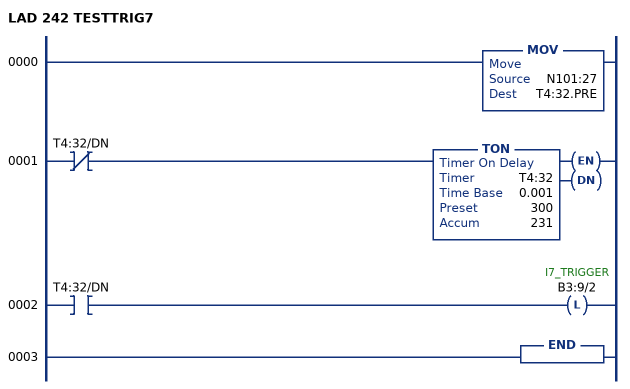
% Rung: 0 %
SOR MOV N101:27 T4:32.PRE EOR
%   N101:27  I7_TRIGTIME %
% Rung: 1 %
SOR XIO T4:32/DN TON T4:32 0.001 300 231 EOR
% Rung: 2 %
SOR XIC T4:32/DN OTL B3:9/2 EOR
%   B3:9/2  I7_TRIGGER %
% Rung: 3 %
SOR END EOR

LADDER 243 "TESTTRIG8"
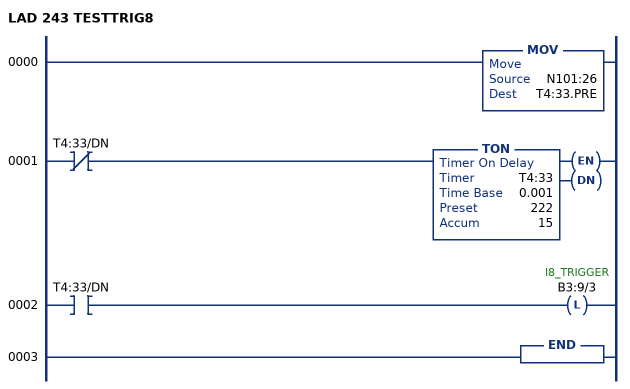
% Rung: 0 %
SOR MOV N101:26 T4:33.PRE EOR
%   N101:26  I8_TRIGTIME %
% Rung: 1 %
SOR XIO T4:33/DN TON T4:33 0.001 222 15 EOR
% Rung: 2 %
SOR XIC T4:33/DN OTL B3:9/3 EOR
%   B3:9/3  I8_TRIGGER %
% Rung: 3 %
SOR END EOR

LADDER 244 "PACKAGER"    % normal %
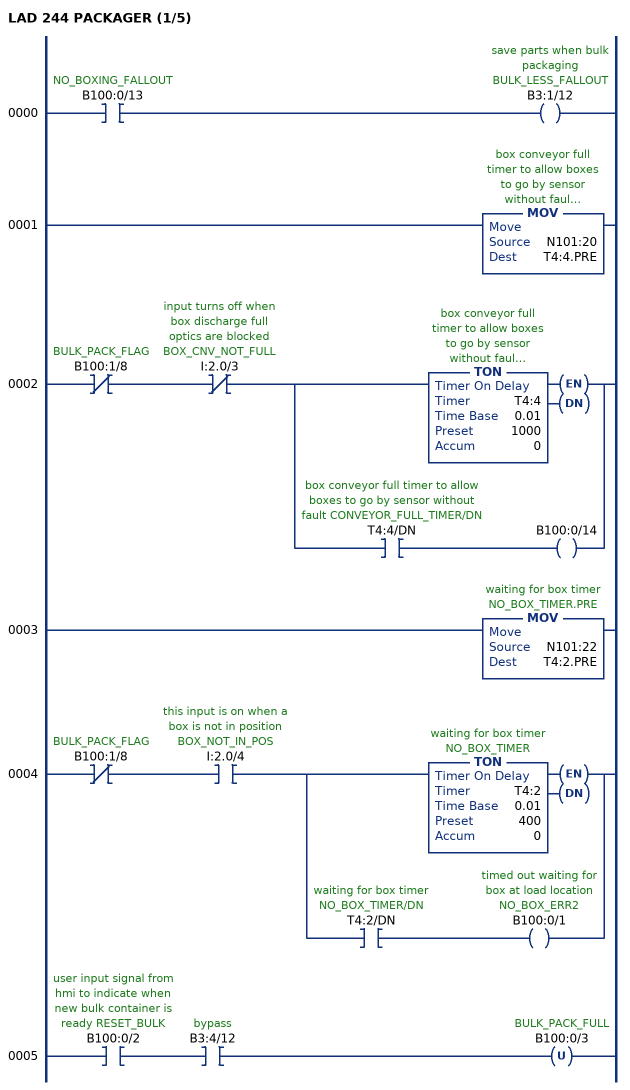
% Rung: 0 %
SOR XIC B100:0/13 OTE B3:1/12 EOR
%   B100:0/13  NO_BOXING_FALLOUT %
%   B3:1/12  BULK_LESS_FALLOUT  "save parts when bulk packaging" %
% Rung: 1 %
SOR MOV N101:20 T4:4.PRE EOR
%   N101:20  CONV_FULL_TIME_LIMIT  "time to allow box to pass box conveyor full sensor without fault" %
%   T4:4  CONVEYOR_FULL_TIMER  "box conveyor full timer to allow boxes to go by sensor without fault" %
% Rung: 2 %
SOR XIO B100:1/8 XIO I:2.0/3 BST TON T4:4 0.01 1000 0 NXB XIC T4:4/DN OTE B100:0/14 BND EOR
%   B100:1/8  BULK_PACK_FLAG %
%   I:2.0/3  BOX_CNV_NOT_FULL  "input turns off when box discharge full optics are blocked" %
%   T4:4  CONVEYOR_FULL_TIMER  "box conveyor full timer to allow boxes to go by sensor without fault" %
% Rung: 3 %
SOR MOV N101:22 T4:2.PRE EOR
%   N101:22  BOX_WAIT_TIME_LIMIT  "the time until waiting for box message in hmi (fault)" %
%   T4:2  NO_BOX_TIMER  "waiting for box timer" %
% Rung: 4 %
SOR XIO B100:1/8 XIC I:2.0/4 BST TON T4:2 0.01 400 0 NXB XIC T4:2/DN OTE B100:0/1 BND EOR
%   B100:1/8  BULK_PACK_FLAG %
%   I:2.0/4  BOX_NOT_IN_POS  "this input is on when a box is not in position" %
%   T4:2  NO_BOX_TIMER  "waiting for box timer" %
%   B100:0/1  NO_BOX_ERR2  "timed out waiting for box at load location" %
% Rung: 5 %
SOR XIC B100:0/2 XIC B3:4/12 OTU B100:0/3 EOR
%   B100:0/2  RESET_BULK  "user input signal from hmi to indicate when new bulk container is ready" %
%   B3:4/12  "bypass" %
%   B100:0/3  BULK_PACK_FULL %

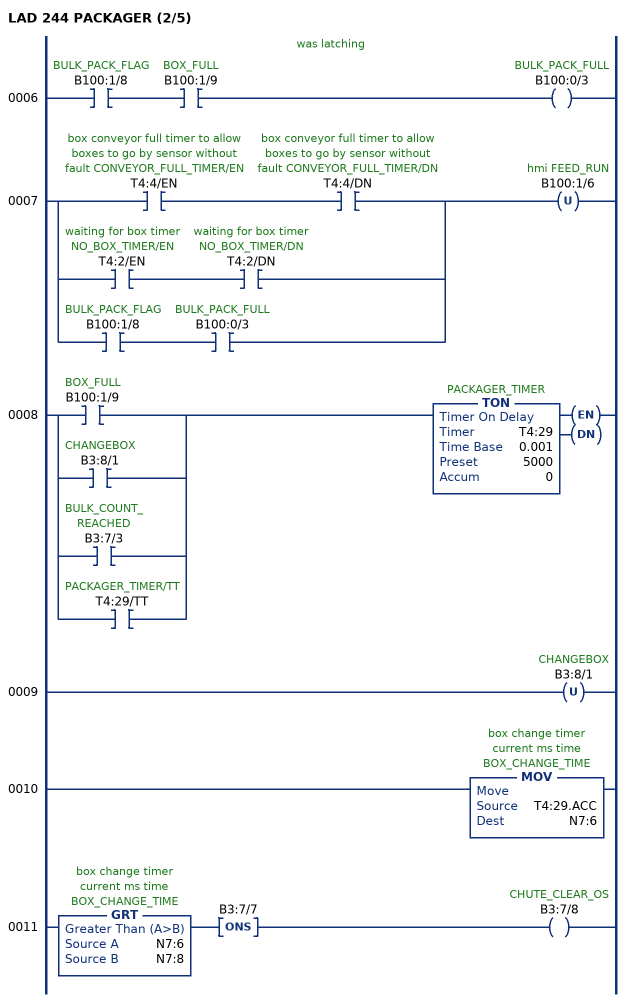
% Rung: 6 %
% was latching %
SOR XIC B100:1/8 XIC B100:1/9 OTE B100:0/3 EOR
%   B100:1/8  BULK_PACK_FLAG %
%   B100:1/9  BOX_FULL %
%   B100:0/3  BULK_PACK_FULL %
% Rung: 7 %
SOR BST XIC T4:4/EN XIC T4:4/DN NXB XIC T4:2/EN XIC T4:2/DN NXB XIC B100:1/8 XIC B100:0/3 BND OTU B100:1/6 EOR
%   T4:4  CONVEYOR_FULL_TIMER  "box conveyor full timer to allow boxes to go by sensor without fault" %
%   T4:2  NO_BOX_TIMER  "waiting for box timer" %
%   B100:1/8  BULK_PACK_FLAG %
%   B100:0/3  BULK_PACK_FULL %
%   B100:1/6  FEED_RUN  "hmi" %
% Rung: 8 %
SOR BST XIC B100:1/9 NXB XIC B3:8/1 NXB XIC B3:7/3 NXB XIC T4:29/TT BND TON T4:29 0.001 5000 0 EOR
%   B100:1/9  BOX_FULL %
%   B3:8/1  CHANGEBOX %
%   B3:7/3  BULK_COUNT_REACHED %
%   T4:29  PACKAGER_TIMER %
% Rung: 9 %
SOR OTU B3:8/1 EOR
%   B3:8/1  CHANGEBOX %
% Rung: 10 %
SOR MOV T4:29.ACC N7:6 EOR
%   T4:29  PACKAGER_TIMER %
%   N7:6  BOX_CHANGE_TIME  "box change timer current ms time" %
% Rung: 11 %
SOR GRT N7:6 N7:8 ONS B3:7/7 OTE B3:7/8 EOR
%   N7:6  BOX_CHANGE_TIME  "box change timer current ms time" %
%   N7:8  CHUTE_CLEAR_TIME %
%   B3:7/8  CHUTE_CLEAR_OS %

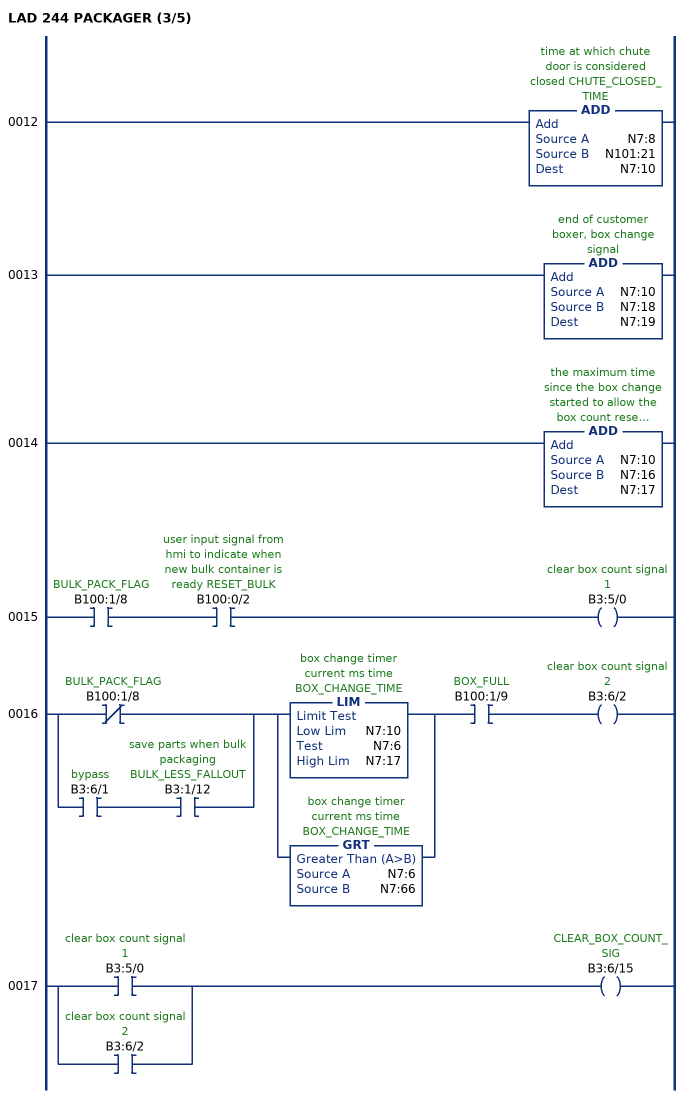
% Rung: 12 %
SOR ADD N7:8 N101:21 N7:10 EOR
%   N7:8  CHUTE_CLEAR_TIME %
%   N101:21  CHUTE_CLOSE_TIME  "ms time required to close chute" %
%   N7:10  CHUTE_CLOSED_TIME  "time at which chute door is considered closed" %
% Rung: 13 %
SOR ADD N7:10 N7:18 N7:19 EOR
%   N7:10  CHUTE_CLOSED_TIME  "time at which chute door is considered closed" %
%   N7:18  CHANGE_BOX_SIG_TIME  "customer boxer change box signal time" %
%   N7:19  "end of customer boxer, box change signal" %
% Rung: 14 %
SOR ADD N7:10 N7:16 N7:17 EOR
%   N7:10  CHUTE_CLOSED_TIME  "time at which chute door is considered closed" %
%   N7:16  RESET_COUNT_SIG_TIME  "maximum length of time to hold box count reset signal on" %
%   N7:17  "the maximum time since the box change started to allow the box count reset signal" %
% Rung: 15 %
SOR XIC B100:1/8 XIC B100:0/2 OTE B3:5/0 EOR
%   B100:1/8  BULK_PACK_FLAG %
%   B100:0/2  RESET_BULK  "user input signal from hmi to indicate when new bulk container is ready" %
%   B3:5/0  "clear box count signal 1" %
% Rung: 16 %
SOR BST XIO B100:1/8 NXB XIC B3:6/1 XIC B3:1/12 BND BST LIM N7:10 N7:6 N7:17 NXB GRT N7:6 N7:66 BND XIC B100:1/9 OTE B3:6/2 EOR
%   B100:1/8  BULK_PACK_FLAG %
%   B3:6/1  "bypass" %
%   B3:1/12  BULK_LESS_FALLOUT  "save parts when bulk packaging" %
%   N7:10  CHUTE_CLOSED_TIME  "time at which chute door is considered closed" %
%   N7:6  BOX_CHANGE_TIME  "box change timer current ms time" %
%   N7:17  "the maximum time since the box change started to allow the box count reset signal" %
%   B100:1/9  BOX_FULL %
%   B3:6/2  "clear box count signal 2" %
% Rung: 17 %
SOR BST XIC B3:5/0 NXB XIC B3:6/2 BND OTE B3:6/15 EOR
%   B3:5/0  "clear box count signal 1" %
%   B3:6/2  "clear box count signal 2" %
%   B3:6/15  CLEAR_BOX_COUNT_SIG %

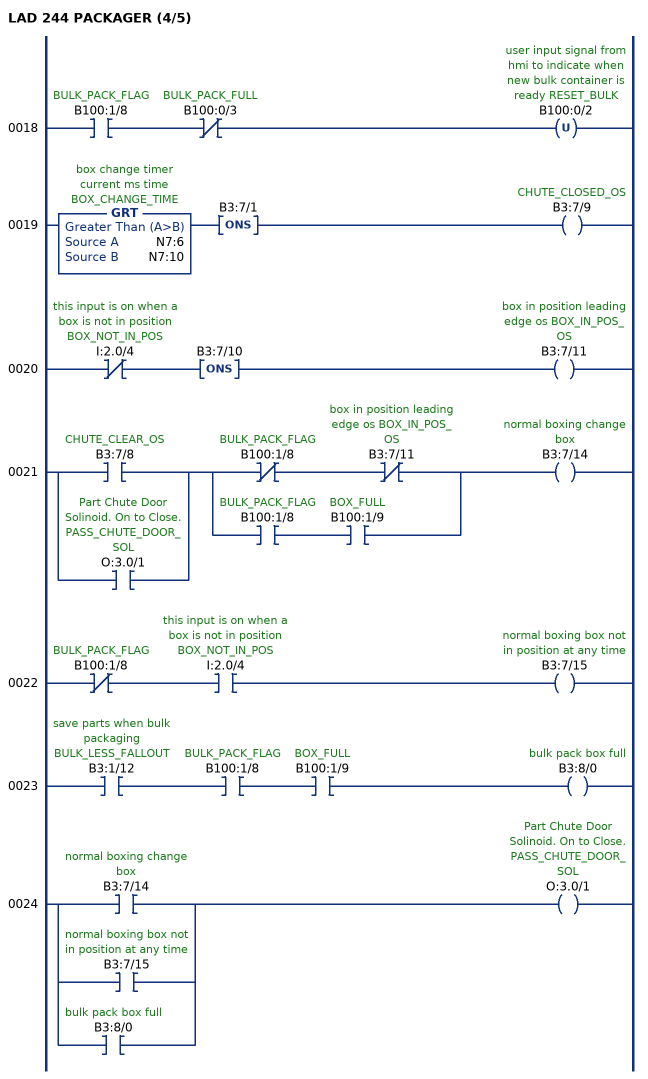
% Rung: 18 %
SOR XIC B100:1/8 XIO B100:0/3 OTU B100:0/2 EOR
%   B100:1/8  BULK_PACK_FLAG %
%   B100:0/3  BULK_PACK_FULL %
%   B100:0/2  RESET_BULK  "user input signal from hmi to indicate when new bulk container is ready" %
% Rung: 19 %
SOR GRT N7:6 N7:10 ONS B3:7/1 OTE B3:7/9 EOR
%   N7:6  BOX_CHANGE_TIME  "box change timer current ms time" %
%   N7:10  CHUTE_CLOSED_TIME  "time at which chute door is considered closed" %
%   B3:7/9  CHUTE_CLOSED_OS %
% Rung: 20 %
SOR XIO I:2.0/4 ONS B3:7/10 OTE B3:7/11 EOR
%   I:2.0/4  BOX_NOT_IN_POS  "this input is on when a box is not in position" %
%   B3:7/11  BOX_IN_POS_OS  "box in position leading edge os" %
% Rung: 21 %
SOR BST XIC B3:7/8 NXB XIC O:3.0/1 BND BST XIO B100:1/8 XIO B3:7/11 NXB XIC B100:1/8 XIC B100:1/9 BND OTE B3:7/14 EOR
%   B3:7/8  CHUTE_CLEAR_OS %
%   O:3.0/1  PASS_CHUTE_DOOR_SOL  "Part Chute Door Solinoid. On to Close." %
%   B100:1/8  BULK_PACK_FLAG %
%   B3:7/11  BOX_IN_POS_OS  "box in position leading edge os" %
%   B100:1/9  BOX_FULL %
%   B3:7/14  "normal boxing change box" %
% Rung: 22 %
SOR XIO B100:1/8 XIC I:2.0/4 OTE B3:7/15 EOR
%   B100:1/8  BULK_PACK_FLAG %
%   I:2.0/4  BOX_NOT_IN_POS  "this input is on when a box is not in position" %
%   B3:7/15  "normal boxing box not in position at any time" %
% Rung: 23 %
SOR XIC B3:1/12 XIC B100:1/8 XIC B100:1/9 OTE B3:8/0 EOR
%   B3:1/12  BULK_LESS_FALLOUT  "save parts when bulk packaging" %
%   B100:1/8  BULK_PACK_FLAG %
%   B100:1/9  BOX_FULL %
%   B3:8/0  "bulk pack box full" %
% Rung: 24 %
SOR BST XIC B3:7/14 NXB XIC B3:7/15 NXB XIC B3:8/0 BND OTE O:3.0/1 EOR
%   B3:7/14  "normal boxing change box" %
%   B3:7/15  "normal boxing box not in position at any time" %
%   B3:8/0  "bulk pack box full" %
%   O:3.0/1  PASS_CHUTE_DOOR_SOL  "Part Chute Door Solinoid. On to Close." %

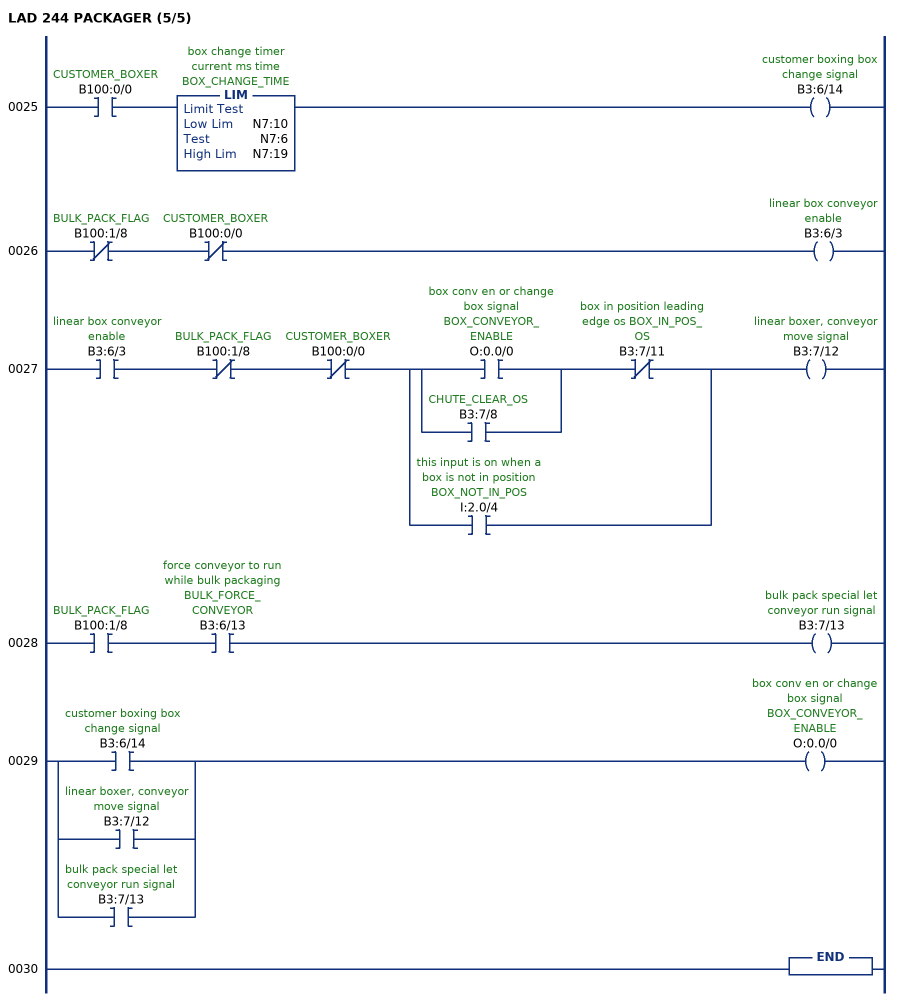
% Rung: 25 %
SOR XIC B100:0/0 LIM N7:10 N7:6 N7:19 OTE B3:6/14 EOR
%   B100:0/0  CUSTOMER_BOXER %
%   N7:10  CHUTE_CLOSED_TIME  "time at which chute door is considered closed" %
%   N7:6  BOX_CHANGE_TIME  "box change timer current ms time" %
%   N7:19  "end of customer boxer, box change signal" %
%   B3:6/14  "customer boxing box change signal" %
% Rung: 26 %
SOR XIO B100:1/8 XIO B100:0/0 OTE B3:6/3 EOR
%   B100:1/8  BULK_PACK_FLAG %
%   B100:0/0  CUSTOMER_BOXER %
%   B3:6/3  "linear box conveyor enable" %
% Rung: 27 %
SOR XIC B3:6/3 XIO B100:1/8 XIO B100:0/0 BST BST XIC O:0.0/0 NXB XIC B3:7/8 BND XIO B3:7/11 NXB XIC I:2.0/4 BND OTE B3:7/12 EOR
%   B3:6/3  "linear box conveyor enable" %
%   B100:1/8  BULK_PACK_FLAG %
%   B100:0/0  CUSTOMER_BOXER %
%   O:0.0/0  BOX_CONVEYOR_ENABLE  "box conv en or change box signal" %
%   B3:7/8  CHUTE_CLEAR_OS %
%   B3:7/11  BOX_IN_POS_OS  "box in position leading edge os" %
%   I:2.0/4  BOX_NOT_IN_POS  "this input is on when a box is not in position" %
%   B3:7/12  "linear boxer, conveyor move signal" %
% Rung: 28 %
SOR XIC B100:1/8 XIC B3:6/13 OTE B3:7/13 EOR
%   B100:1/8  BULK_PACK_FLAG %
%   B3:6/13  BULK_FORCE_CONVEYOR  "force conveyor to run while bulk packaging" %
%   B3:7/13  "bulk pack special let conveyor run signal" %
% Rung: 29 %
SOR BST XIC B3:6/14 NXB XIC B3:7/12 NXB XIC B3:7/13 BND OTE O:0.0/0 EOR
%   B3:6/14  "customer boxing box change signal" %
%   B3:7/12  "linear boxer, conveyor move signal" %
%   B3:7/13  "bulk pack special let conveyor run signal" %
%   O:0.0/0  BOX_CONVEYOR_ENABLE  "box conv en or change box signal" %
% Rung: 30 %
SOR END EOR

LADDER 245 "NO PACKAGE"
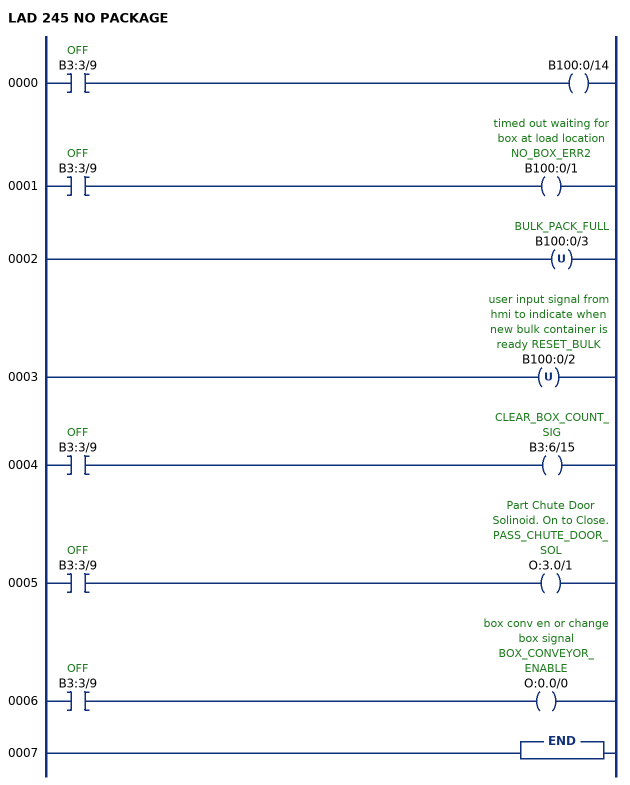
% Rung: 0 %
SOR XIC B3:3/9 OTE B100:0/14 EOR
%   B3:3/9  OFF %
% Rung: 1 %
SOR XIC B3:3/9 OTE B100:0/1 EOR
%   B3:3/9  OFF %
%   B100:0/1  NO_BOX_ERR2  "timed out waiting for box at load location" %
% Rung: 2 %
SOR OTU B100:0/3 EOR
%   B100:0/3  BULK_PACK_FULL %
% Rung: 3 %
SOR OTU B100:0/2 EOR
%   B100:0/2  RESET_BULK  "user input signal from hmi to indicate when new bulk container is ready" %
% Rung: 4 %
SOR XIC B3:3/9 OTE B3:6/15 EOR
%   B3:3/9  OFF %
%   B3:6/15  CLEAR_BOX_COUNT_SIG %
% Rung: 5 %
SOR XIC B3:3/9 OTE O:3.0/1 EOR
%   B3:3/9  OFF %
%   O:3.0/1  PASS_CHUTE_DOOR_SOL  "Part Chute Door Solinoid. On to Close." %
% Rung: 6 %
SOR XIC B3:3/9 OTE O:0.0/0 EOR
%   B3:3/9  OFF %
%   O:0.0/0  BOX_CONVEYOR_ENABLE  "box conv en or change box signal" %
% Rung: 7 %
SOR END EOR

LADDER 246 "RATE1"
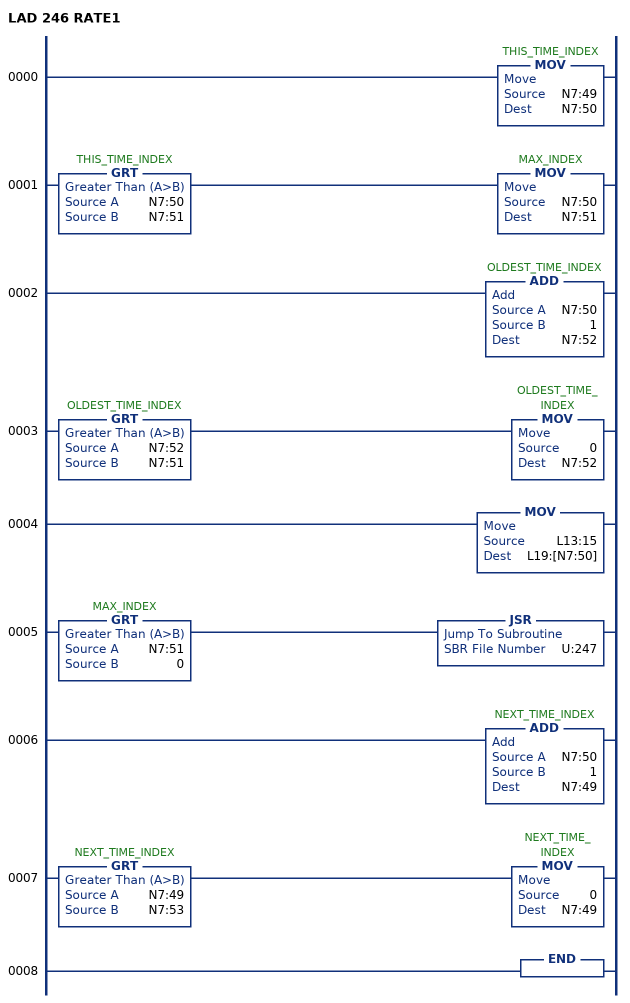
% Rung: 0 %
SOR MOV N7:49 N7:50 EOR
%   N7:49  NEXT_TIME_INDEX %
%   N7:50  THIS_TIME_INDEX %
% Rung: 1 %
SOR GRT N7:50 N7:51 MOV N7:50 N7:51 EOR
%   N7:50  THIS_TIME_INDEX %
%   N7:51  MAX_INDEX %
% Rung: 2 %
SOR ADD N7:50 1 N7:52 EOR
%   N7:50  THIS_TIME_INDEX %
%   N7:52  OLDEST_TIME_INDEX %
% Rung: 3 %
SOR GRT N7:52 N7:51 MOV 0 N7:52 EOR
%   N7:52  OLDEST_TIME_INDEX %
%   N7:51  MAX_INDEX %
% Rung: 4 %
SOR MOV L13:15 L19:[N7:50] EOR
%   L13:15  THE_TIME %
%   N7:50  THIS_TIME_INDEX %
% Rung: 5 %
SOR GRT N7:51 0 JSR U:247 EOR
%   N7:51  MAX_INDEX %
% Rung: 6 %
SOR ADD N7:50 1 N7:49 EOR
%   N7:50  THIS_TIME_INDEX %
%   N7:49  NEXT_TIME_INDEX %
% Rung: 7 %
SOR GRT N7:49 N7:53 MOV 0 N7:49 EOR
%   N7:49  NEXT_TIME_INDEX %
%   N7:53  UPPER_INDEX_LIMIT %
% Rung: 8 %
SOR END EOR

LADDER 247 "RATE2"
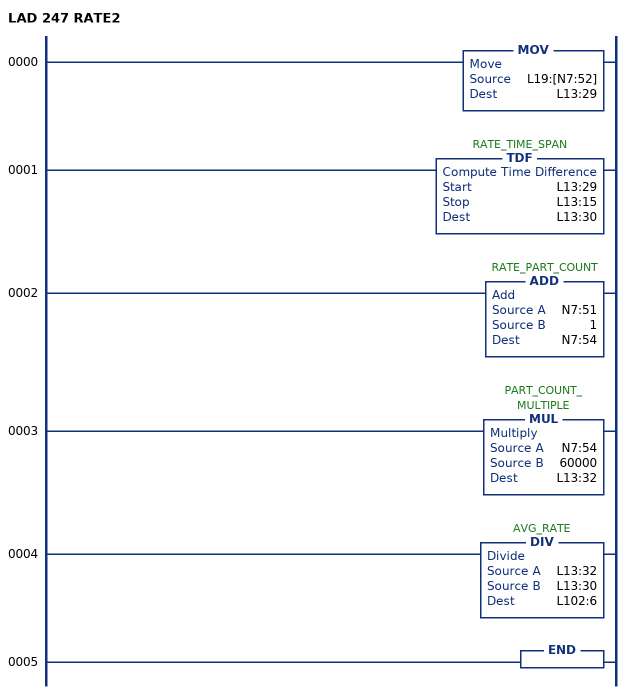
% Rung: 0 %
SOR MOV L19:[N7:52] L13:29 EOR
%   N7:52  OLDEST_TIME_INDEX %
% Rung: 1 %
SOR TDF L13:29 L13:15 L13:30 EOR
%   L13:15  THE_TIME %
%   L13:30  RATE_TIME_SPAN %
% Rung: 2 %
SOR ADD N7:51 1 N7:54 EOR
%   N7:51  MAX_INDEX %
%   N7:54  RATE_PART_COUNT %
% Rung: 3 %
SOR MUL N7:54 60000 L13:32 EOR
%   N7:54  RATE_PART_COUNT %
%   L13:32  PART_COUNT_MULTIPLE %
% Rung: 4 %
SOR DIV L13:32 L13:30 L102:6 EOR
%   L13:32  PART_COUNT_MULTIPLE %
%   L13:30  RATE_TIME_SPAN %
%   L102:6  AVG_RATE %
% Rung: 5 %
SOR END EOR

LADDER 248 "RESET RATE"
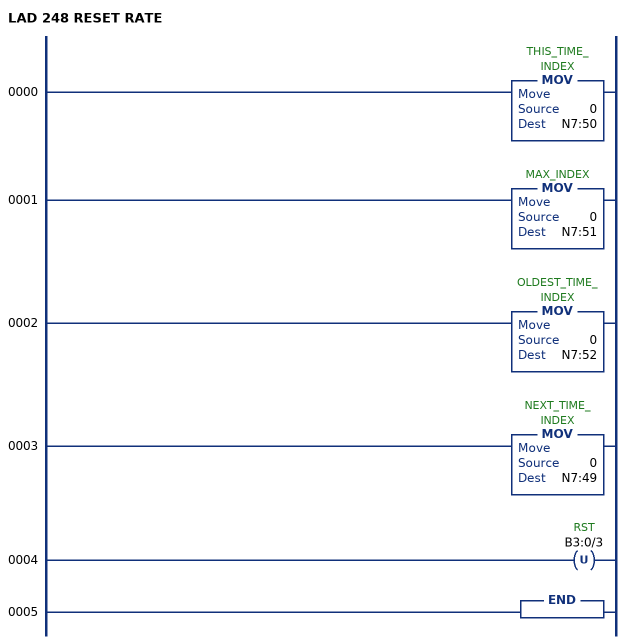
% Rung: 0 %
SOR MOV 0 N7:50 EOR
%   N7:50  THIS_TIME_INDEX %
% Rung: 1 %
SOR MOV 0 N7:51 EOR
%   N7:51  MAX_INDEX %
% Rung: 2 %
SOR MOV 0 N7:52 EOR
%   N7:52  OLDEST_TIME_INDEX %
% Rung: 3 %
SOR MOV 0 N7:49 EOR
%   N7:49  NEXT_TIME_INDEX %
% Rung: 4 %
SOR OTU B3:0/3 EOR
%   B3:0/3  RST %
% Rung: 5 %
SOR END EOR

LADDER 249 "NP STOP"    % stop on no good %
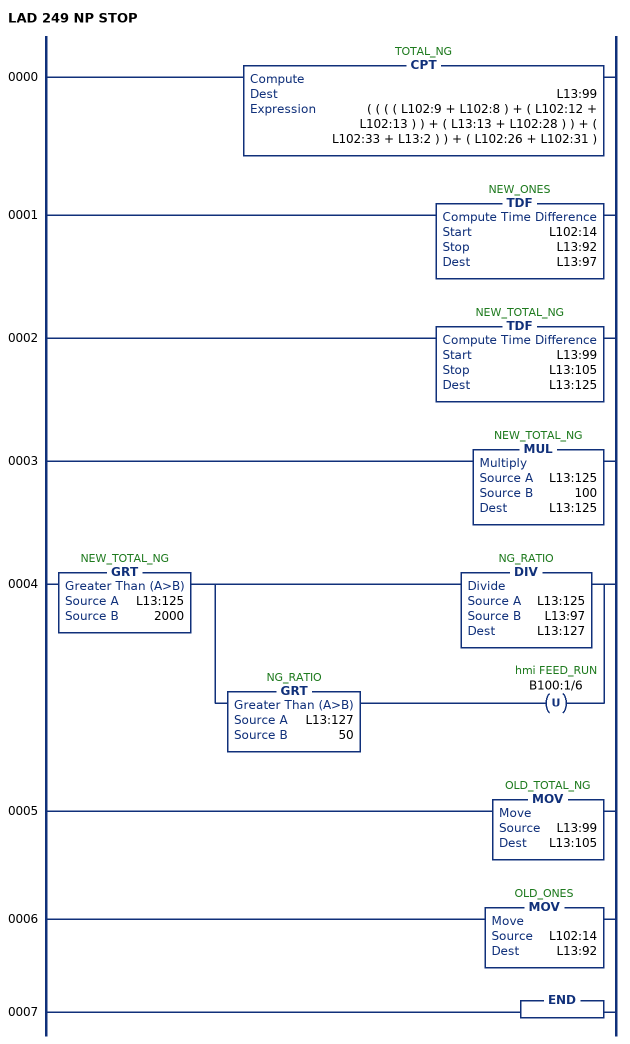
% Rung: 0 %
SOR CPT L13:99 " ( ( ( ( L102:9 + L102:8 ) + ( L102:12 + L102:13 ) ) + ( L13:13 + L102:28 ) ) + ( L102:33 + L13:2 ) ) + ( L102:26 + L102:31 ) " EOR
%   L13:99  TOTAL_NG %
%   L102:9  "too wide bottom" %
%   L102:8  "too close bottom" %
%   L102:12  "too close top count" %
%   L102:13  "too wide top count" %
%   L102:28  I1_I5_SKIPPEDCOUNT %
%   L102:33  I2_I6_SKIPPEDCOUNT %
%   L102:26  I1_I5_FAIL_COUNT %
%   L102:31  I2_I6_FAIL_COUNT %
% Rung: 1 %
SOR TDF L102:14 L13:92 L13:97 EOR
%   L102:14  ONES %
%   L13:92  OLD_ONES %
%   L13:97  NEW_ONES %
% Rung: 2 %
SOR TDF L13:99 L13:105 L13:125 EOR
%   L13:99  TOTAL_NG %
%   L13:105  OLD_TOTAL_NG %
%   L13:125  NEW_TOTAL_NG %
% Rung: 3 %
SOR MUL L13:125 100 L13:125 EOR
%   L13:125  NEW_TOTAL_NG %
% Rung: 4 %
SOR GRT L13:125 2000 BST DIV L13:125 L13:97 L13:127 NXB GRT L13:127 50 OTU B100:1/6 BND EOR
%   L13:125  NEW_TOTAL_NG %
%   L13:97  NEW_ONES %
%   L13:127  NG_RATIO %
%   B100:1/6  FEED_RUN  "hmi" %
% Rung: 5 %
SOR MOV L13:99 L13:105 EOR
%   L13:99  TOTAL_NG %
%   L13:105  OLD_TOTAL_NG %
% Rung: 6 %
SOR MOV L102:14 L13:92 EOR
%   L102:14  ONES %
%   L13:92  OLD_ONES %
% Rung: 7 %
SOR END EOR

LADDER 250 "SPEED BOT"    % high speed %
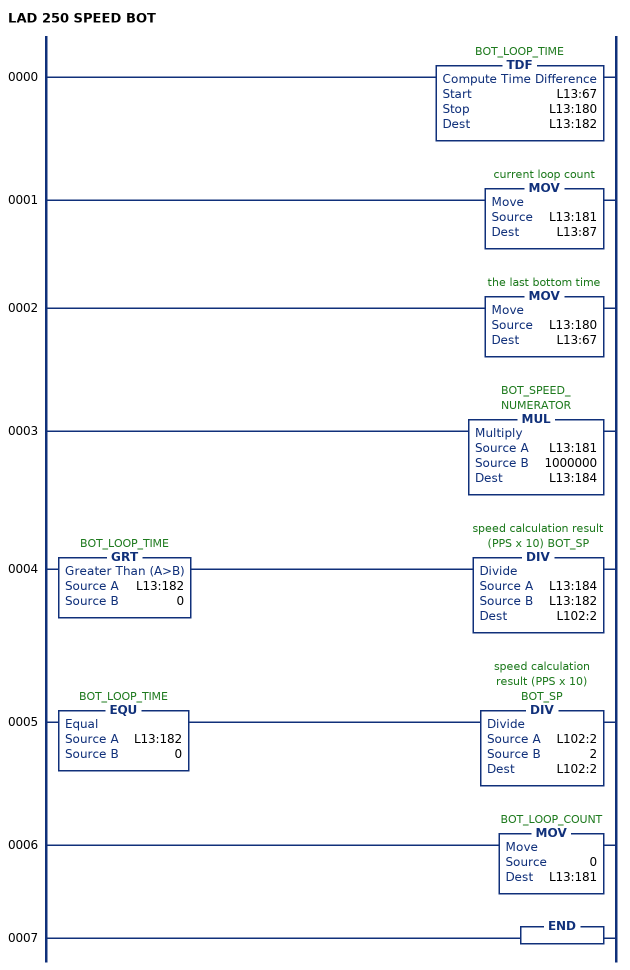
% Rung: 0 %
SOR TDF L13:67 L13:180 L13:182 EOR
%   L13:67  "the last bottom time" %
%   L13:180  BOT_THIS_TIME  "rtc bot belt movement event time" %
%   L13:182  BOT_LOOP_TIME %
% Rung: 1 %
SOR MOV L13:181 L13:87 EOR
%   L13:181  BOT_LOOP_COUNT %
%   L13:87  "current loop count" %
% Rung: 2 %
SOR MOV L13:180 L13:67 EOR
%   L13:180  BOT_THIS_TIME  "rtc bot belt movement event time" %
%   L13:67  "the last bottom time" %
% Rung: 3 %
SOR MUL L13:181 1000000 L13:184 EOR
%   L13:181  BOT_LOOP_COUNT %
%   L13:184  BOT_SPEED_NUMERATOR %
% Rung: 4 %
SOR GRT L13:182 0 DIV L13:184 L13:182 L102:2 EOR
%   L13:182  BOT_LOOP_TIME %
%   L13:184  BOT_SPEED_NUMERATOR %
%   L102:2  BOT_SP  "speed calculation result (PPS x 10)" %
% Rung: 5 %
SOR EQU L13:182 0 DIV L102:2 2 L102:2 EOR
%   L13:182  BOT_LOOP_TIME %
%   L102:2  BOT_SP  "speed calculation result (PPS x 10)" %
% Rung: 6 %
SOR MOV 0 L13:181 EOR
%   L13:181  BOT_LOOP_COUNT %
% Rung: 7 %
SOR END EOR

LADDER 251 "SPEED TOP"    % high speed %
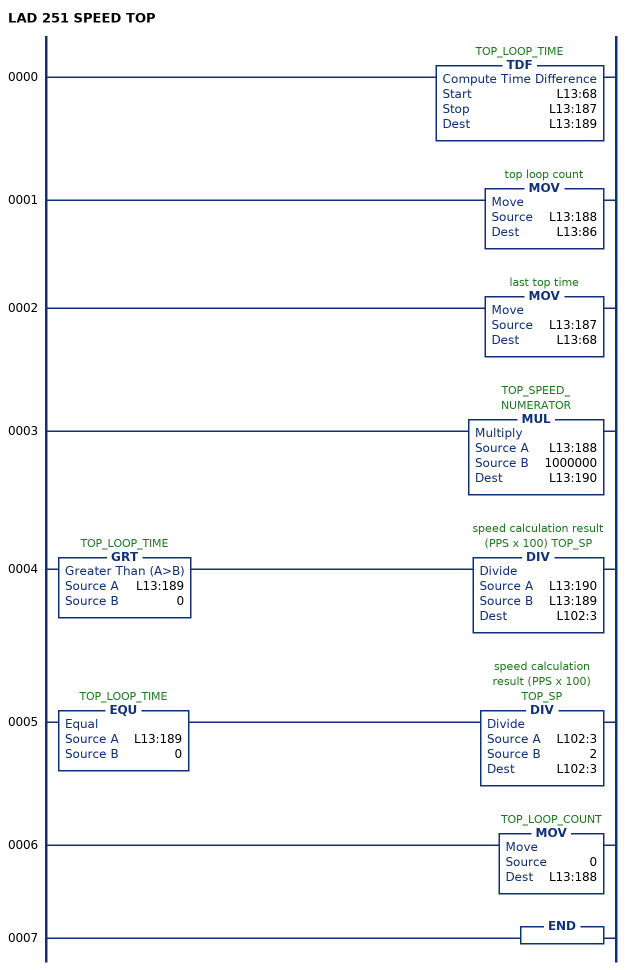
% Rung: 0 %
SOR TDF L13:68 L13:187 L13:189 EOR
%   L13:68  "last top time" %
%   L13:187  TOP_THIS_TIME  "rtc top belt movement event time" %
%   L13:189  TOP_LOOP_TIME %
% Rung: 1 %
SOR MOV L13:188 L13:86 EOR
%   L13:188  TOP_LOOP_COUNT %
%   L13:86  "top loop count" %
% Rung: 2 %
SOR MOV L13:187 L13:68 EOR
%   L13:187  TOP_THIS_TIME  "rtc top belt movement event time" %
%   L13:68  "last top time" %
% Rung: 3 %
SOR MUL L13:188 1000000 L13:190 EOR
%   L13:188  TOP_LOOP_COUNT %
%   L13:190  TOP_SPEED_NUMERATOR %
% Rung: 4 %
SOR GRT L13:189 0 DIV L13:190 L13:189 L102:3 EOR
%   L13:189  TOP_LOOP_TIME %
%   L13:190  TOP_SPEED_NUMERATOR %
%   L102:3  TOP_SP  "speed calculation result (PPS x 100)" %
% Rung: 5 %
SOR EQU L13:189 0 DIV L102:3 2 L102:3 EOR
%   L13:189  TOP_LOOP_TIME %
%   L102:3  TOP_SP  "speed calculation result (PPS x 100)" %
% Rung: 6 %
SOR MOV 0 L13:188 EOR
%   L13:188  TOP_LOOP_COUNT %
% Rung: 7 %
SOR END EOR

LADDER 252 "P BOT"    % high speed %
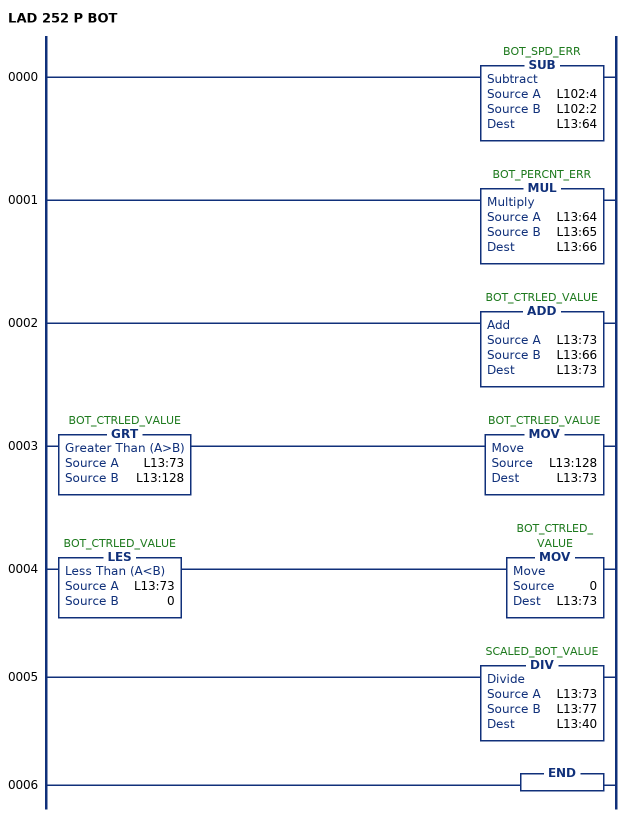
% Rung: 0 %
SOR SUB L102:4 L102:2 L13:64 EOR
%   L102:4  BOT_SPD_SETPOINT %
%   L102:2  BOT_SP  "speed calculation result (PPS x 10)" %
%   L13:64  BOT_SPD_ERR %
% Rung: 1 %
SOR MUL L13:64 L13:65 L13:66 EOR
%   L13:64  BOT_SPD_ERR %
%   L13:65  POS5SHIFT %
%   L13:66  BOT_PERCNT_ERR %
% Rung: 2 %
SOR ADD L13:73 L13:66 L13:73 EOR
%   L13:73  BOT_CTRLED_VALUE %
%   L13:66  BOT_PERCNT_ERR %
% Rung: 3 %
SOR GRT L13:73 L13:128 MOV L13:128 L13:73 EOR
%   L13:73  BOT_CTRLED_VALUE %
%   L13:128  "how much top has shifted since measurment" %
% Rung: 4 %
SOR LES L13:73 0 MOV 0 L13:73 EOR
%   L13:73  BOT_CTRLED_VALUE %
% Rung: 5 %
SOR DIV L13:73 L13:77 L13:40 EOR
%   L13:73  BOT_CTRLED_VALUE %
%   L13:40  SCALED_BOT_VALUE %
% Rung: 6 %
SOR END EOR

LADDER 253 "P TOP"    % high speed %
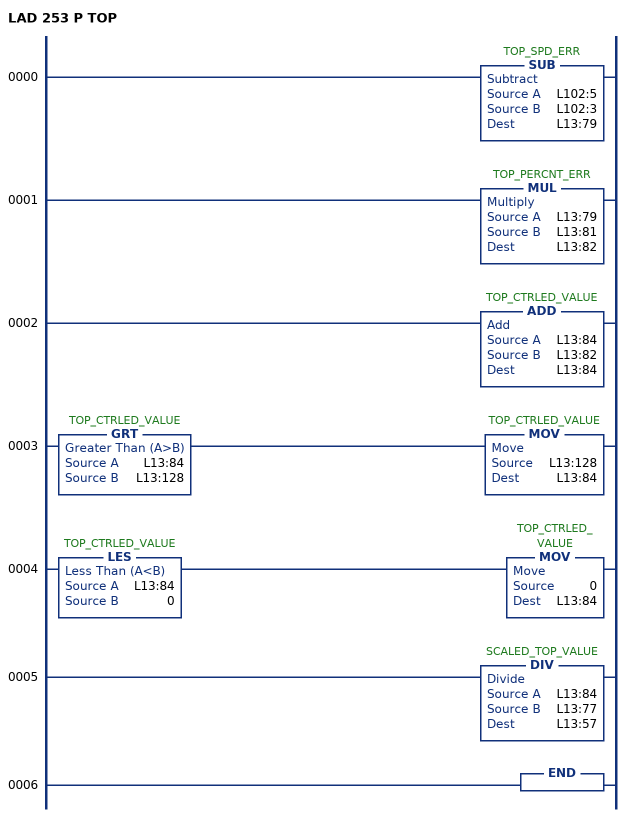
% Rung: 0 %
SOR SUB L102:5 L102:3 L13:79 EOR
%   L102:5  TOP_SPD_SETPOINT %
%   L102:3  TOP_SP  "speed calculation result (PPS x 100)" %
%   L13:79  TOP_SPD_ERR %
% Rung: 1 %
SOR MUL L13:79 L13:81 L13:82 EOR
%   L13:79  TOP_SPD_ERR %
%   L13:81  TOP_FDBK_RATIO %
%   L13:82  TOP_PERCNT_ERR %
% Rung: 2 %
SOR ADD L13:84 L13:82 L13:84 EOR
%   L13:84  TOP_CTRLED_VALUE %
%   L13:82  TOP_PERCNT_ERR %
% Rung: 3 %
SOR GRT L13:84 L13:128 MOV L13:128 L13:84 EOR
%   L13:84  TOP_CTRLED_VALUE %
%   L13:128  "how much top has shifted since measurment" %
% Rung: 4 %
SOR LES L13:84 0 MOV 0 L13:84 EOR
%   L13:84  TOP_CTRLED_VALUE %
% Rung: 5 %
SOR DIV L13:84 L13:77 L13:57 EOR
%   L13:84  TOP_CTRLED_VALUE %
%   L13:57  SCALED_TOP_VALUE %
% Rung: 6 %
SOR END EOR

LADDER 254 "TOTALCOUNT"
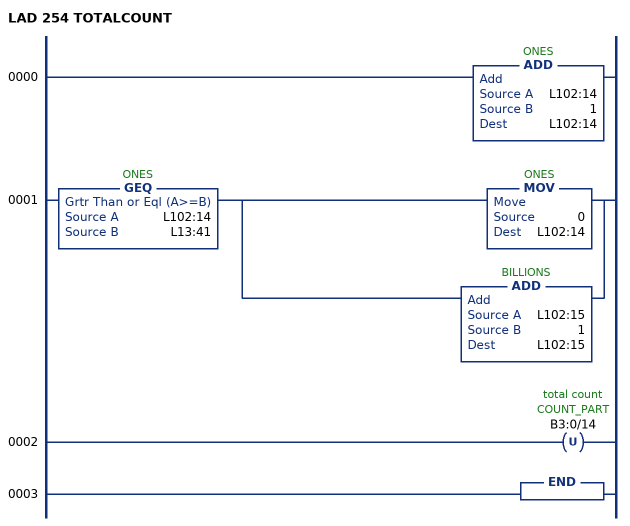
% Rung: 0 %
SOR ADD L102:14 1 L102:14 EOR
%   L102:14  ONES %
% Rung: 1 %
SOR GEQ L102:14 L13:41 BST MOV 0 L102:14 NXB ADD L102:15 1 L102:15 BND EOR
%   L102:14  ONES %
%   L13:41  "skipped count change in the last 3 seconds" %
%   L102:15  BILLIONS %
% Rung: 2 %
SOR OTU B3:0/14 EOR
%   B3:0/14  COUNT_PART  "total count" %
% Rung: 3 %
SOR END EOR

LADDER 255 "SAVED"
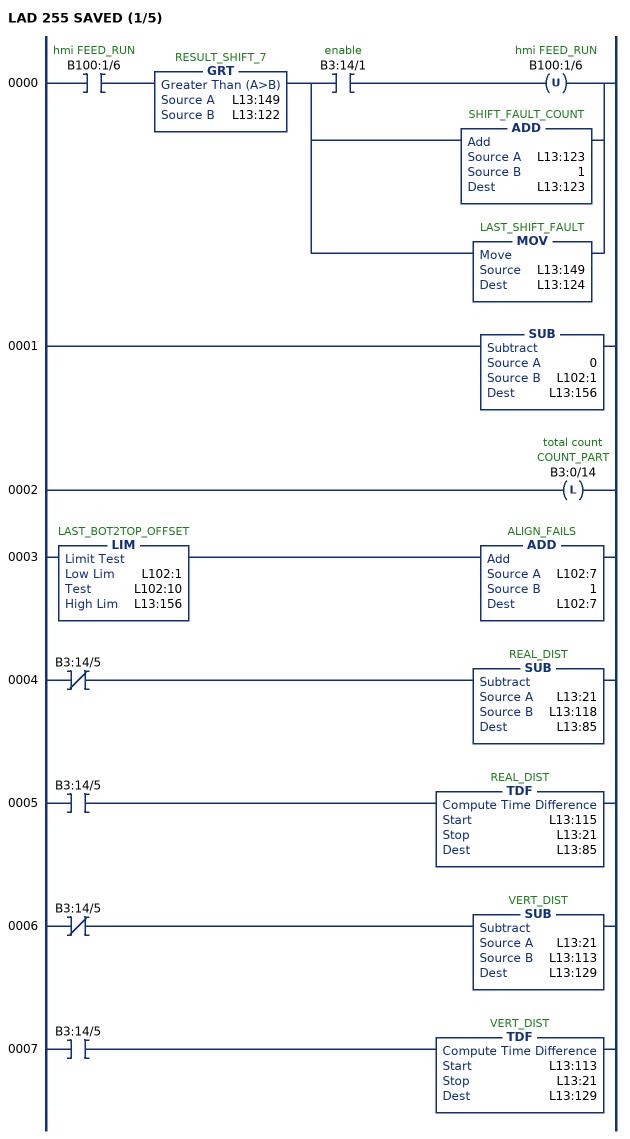
% Rung: 0 %
SOR XIC B100:1/6 GRT L13:149 L13:122 BST XIC B3:14/1 OTU B100:1/6 NXB ADD L13:123 1 L13:123 NXB MOV L13:149 L13:124 BND EOR
%   B100:1/6  FEED_RUN  "hmi" %
%   L13:149  RESULT_SHIFT_7 %
%   L13:122  TOP_SHIFT_FAULT_LIM  "remove me" %
%   B3:14/1  "enable" %
%   L13:123  SHIFT_FAULT_COUNT %
%   L13:124  LAST_SHIFT_FAULT %
% Rung: 1 %
SOR SUB 0 L102:1 L13:156 EOR
%   L102:1  MAX_OFFSET  "transition zone width" %
% Rung: 2 %
SOR OTL B3:0/14 EOR
%   B3:0/14  COUNT_PART  "total count" %
% Rung: 3 %
SOR LIM L102:1 L102:10 L13:156 ADD L102:7 1 L102:7 EOR
%   L102:1  MAX_OFFSET  "transition zone width" %
%   L102:10  LAST_BOT2TOP_OFFSET %
%   L102:7  ALIGN_FAILS %
% Rung: 4 %
SOR XIO B3:14/5 SUB L13:21 L13:118 L13:85 EOR
%   L13:21  TOP_POSITION %
%   L13:118  REAL_CL_POSITION  "real part center line in raw position" %
%   L13:85  REAL_DIST %
% Rung: 5 %
SOR XIC B3:14/5 TDF L13:115 L13:21 L13:85 EOR
%   L13:115  TRAILING_EDGE_POS  "top optic trailing edge position" %
%   L13:21  TOP_POSITION %
%   L13:85  REAL_DIST %
% Rung: 6 %
SOR XIO B3:14/5 SUB L13:21 L13:113 L13:129 EOR
%   L13:21  TOP_POSITION %
%   L13:113  VIRT_CL_POSITION  "virtual part center line transfer from the bottom in raw position" %
%   L13:129  VERT_DIST %
% Rung: 7 %
SOR XIC B3:14/5 TDF L13:113 L13:21 L13:129 EOR
%   L13:113  VIRT_CL_POSITION  "virtual part center line transfer from the bottom in raw position" %
%   L13:21  TOP_POSITION %
%   L13:129  VERT_DIST %

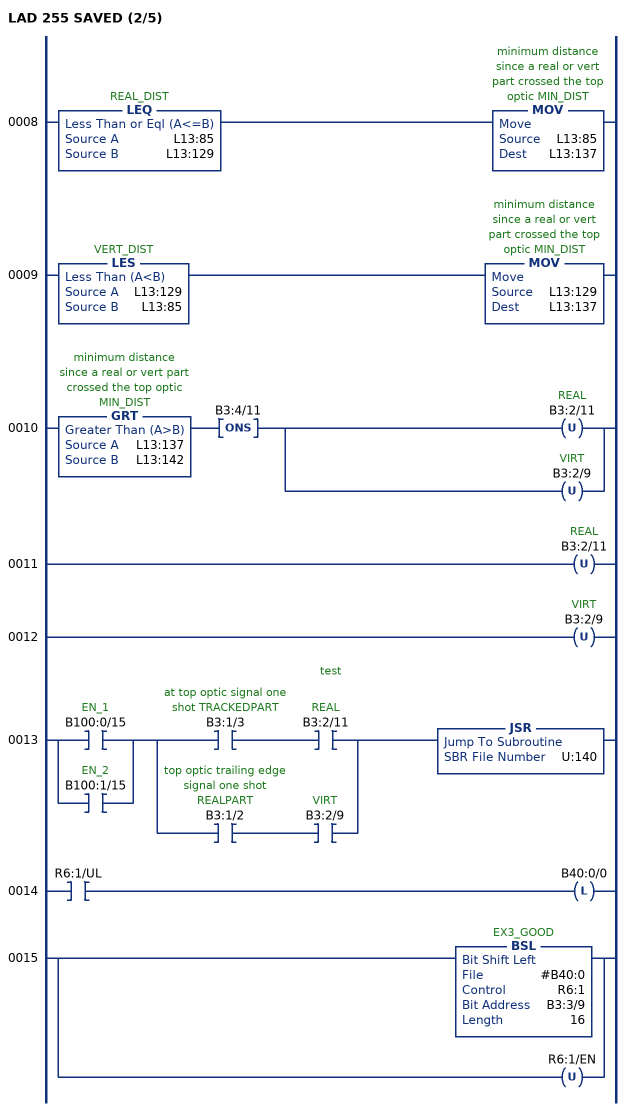
% Rung: 8 %
SOR LEQ L13:85 L13:129 MOV L13:85 L13:137 EOR
%   L13:85  REAL_DIST %
%   L13:129  VERT_DIST %
%   L13:137  MIN_DIST  "minimum distance since a real or vert part crossed the top optic" %
% Rung: 9 %
SOR LES L13:129 L13:85 MOV L13:129 L13:137 EOR
%   L13:129  VERT_DIST %
%   L13:85  REAL_DIST %
%   L13:137  MIN_DIST  "minimum distance since a real or vert part crossed the top optic" %
% Rung: 10 %
SOR GRT L13:137 L13:142 ONS B3:4/11 BST OTU B3:2/11 NXB OTU B3:2/9 BND EOR
%   L13:137  MIN_DIST  "minimum distance since a real or vert part crossed the top optic" %
%   L13:142  LAST_ALIGNMENT_FAILS %
%   B3:2/11  REAL %
%   B3:2/9  VIRT %
% Rung: 11 %
SOR OTU B3:2/11 EOR
%   B3:2/11  REAL %
% Rung: 12 %
SOR OTU B3:2/9 EOR
%   B3:2/9  VIRT %
% Rung: 13 %
% test %
SOR BST XIC B100:0/15 NXB XIC B100:1/15 BND BST XIC B3:1/3 XIC B3:2/11 NXB XIC B3:1/2 XIC B3:2/9 BND JSR U:140 EOR
%   B100:0/15  EN_1 %
%   B100:1/15  EN_2 %
%   B3:1/3  TRACKEDPART  "at top optic signal one shot" %
%   B3:2/11  REAL %
%   B3:1/2  REALPART  "top optic trailing edge signal one shot" %
%   B3:2/9  VIRT %
% Rung: 14 %
SOR XIC R6:1/UL OTL B40:0/0 EOR
% Rung: 15 %
SOR BST BSL #B40:0 R6:1 B3:3/9 16 NXB OTU R6:1/EN BND EOR
%   B40:0  EX3_GOOD %
%   B3:3/9  OFF %

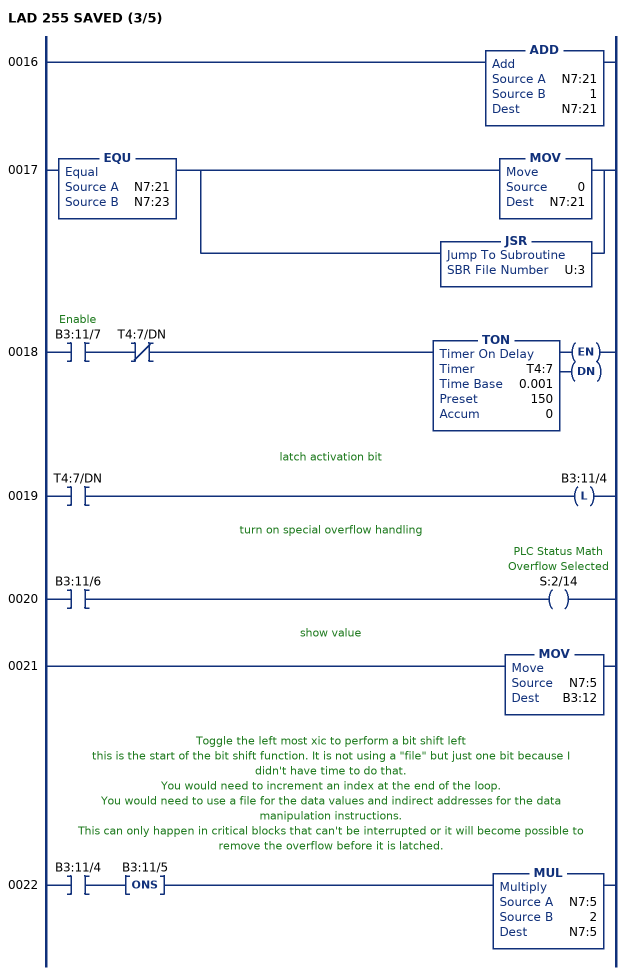
% Rung: 16 %
SOR ADD N7:21 1 N7:21 EOR
% Rung: 17 %
SOR EQU N7:21 N7:23 BST MOV 0 N7:21 NXB JSR U:3 BND EOR
% Rung: 18 %
SOR XIC B3:11/7 XIO T4:7/DN TON T4:7 0.001 150 0 EOR
%   B3:11/7  "Enable" %
% Rung: 19 %
% latch activation bit %
SOR XIC T4:7/DN OTL B3:11/4 EOR
% Rung: 20 %
% turn on special overflow handling %
SOR XIC B3:11/6 OTE S:2/14 EOR
%   S:2/14  "PLC Status Math Overflow Selected" %
% Rung: 21 %
% show value %
SOR MOV N7:5 B3:12 EOR
% Rung: 22 %
% Toggle the left most xic to perform a bit shift left
% 
% this is the start of the bit shift function. It is not using a "file" but just one bit because I didn't have time to do that.
% You would need to increment an index at the end of the loop.
% You would need to use a file for the data values and indirect addresses for the data manipulation instructions.
% 
% This can only happen in critical blocks that can't be interrupted or it will become possible to remove the overflow before it is latched. %
SOR XIC B3:11/4 ONS B3:11/5 MUL N7:5 2 N7:5 EOR

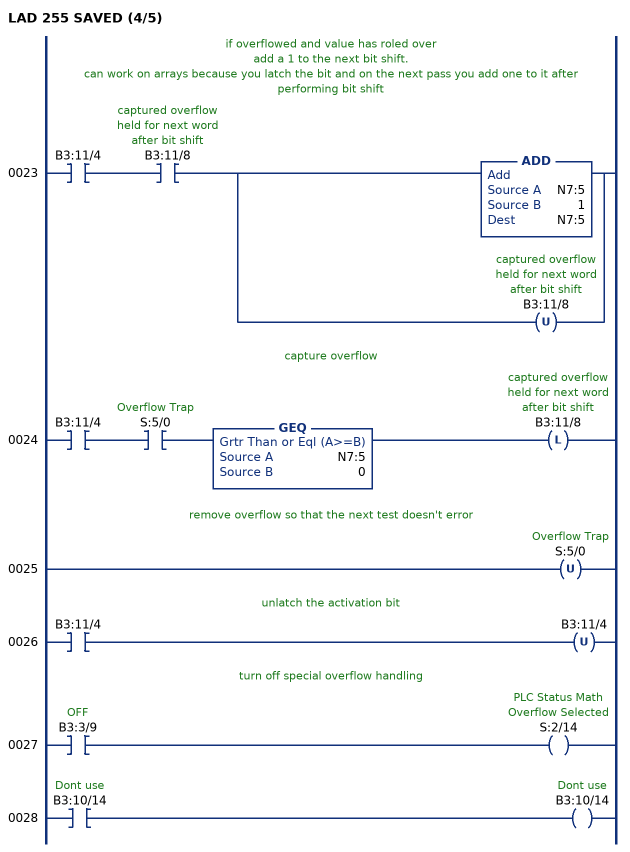
% Rung: 23 %
% if overflowed and value has roled over
% add a 1 to the next bit shift.
% can work on arrays because you latch the bit and on the next pass you add one to it after performing bit shift %
SOR XIC B3:11/4 XIC B3:11/8 BST ADD N7:5 1 N7:5 NXB OTU B3:11/8 BND EOR
%   B3:11/8  "captured overflow held for next word after bit shift" %
% Rung: 24 %
% capture overflow %
SOR XIC B3:11/4 XIC S:5/0 GEQ N7:5 0 OTL B3:11/8 EOR
%   S:5/0  "Overflow Trap" %
%   B3:11/8  "captured overflow held for next word after bit shift" %
% Rung: 25 %
% remove overflow so that the next test doesn't error %
SOR OTU S:5/0 EOR
%   S:5/0  "Overflow Trap" %
% Rung: 26 %
% unlatch the activation bit %
SOR XIC B3:11/4 OTU B3:11/4 EOR
% Rung: 27 %
% turn off special overflow handling %
SOR XIC B3:3/9 OTE S:2/14 EOR
%   B3:3/9  OFF %
%   S:2/14  "PLC Status Math Overflow Selected" %
% Rung: 28 %
SOR XIC B3:10/14 OTE B3:10/14 EOR
%   B3:10/14  "Dont use" %

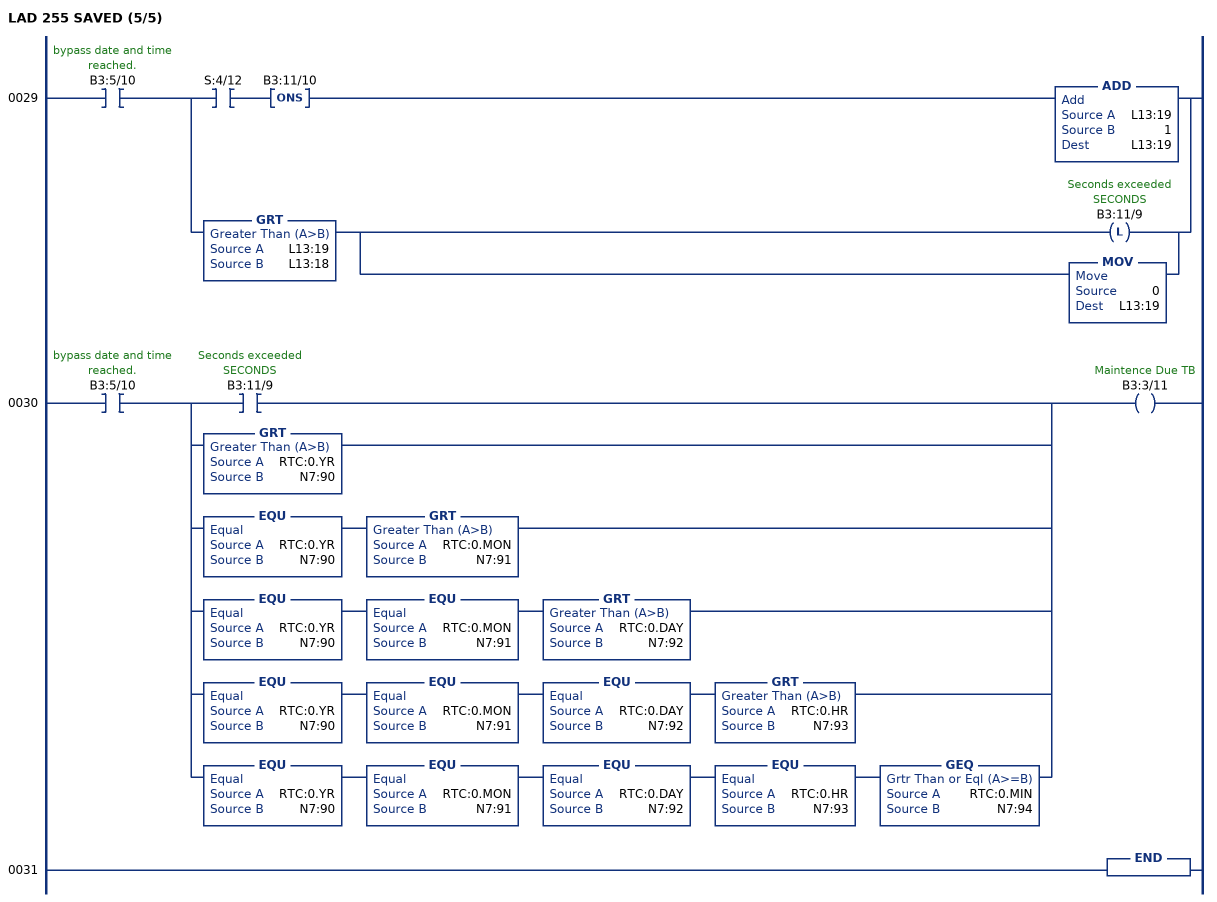
% Rung: 29 %
SOR XIC B3:5/10 BST XIC S:4/12 ONS B3:11/10 ADD L13:19 1 L13:19 NXB GRT L13:19 L13:18 BST OTL B3:11/9 NXB MOV 0 L13:19 BND BND EOR
%   B3:5/10  "bypass date and time reached." %
%   L13:18  MAX %
%   B3:11/9  SECONDS  "Seconds exceeded" %
% Rung: 30 %
SOR XIC B3:5/10 BST XIC B3:11/9 NXB GRT RTC:0.YR N7:90 NXB EQU RTC:0.YR N7:90 GRT RTC:0.MON N7:91 NXB EQU RTC:0.YR N7:90 EQU RTC:0.MON N7:91 GRT RTC:0.DAY N7:92 NXB EQU RTC:0.YR N7:90 EQU RTC:0.MON N7:91 EQU RTC:0.DAY N7:92 GRT RTC:0.HR N7:93 NXB EQU RTC:0.YR N7:90 EQU RTC:0.MON N7:91 EQU RTC:0.DAY N7:92 EQU RTC:0.HR N7:93 GEQ RTC:0.MIN N7:94 BND OTE B3:3/11 EOR
%   B3:5/10  "bypass date and time reached." %
%   B3:11/9  SECONDS  "Seconds exceeded" %
%   N7:90  RTC %
%   B3:3/11  TB  "Maintence Due" %
% Rung: 31 %
SOR END EOR

OTHER DOCUMENTED ADDRESSES
  B3:10/5  "ins 7 pass location okay"
  B3:10/6  "ins 8 pass location okay"
  B3:10/7  "ins 7 passable"
  B3:10/8  "ins 8 passable"
  B38:0  EX1_GOOD
  B189:0/0  "change box"
  B189:0/9  "override boxing ok or not full signal"
  B189:0/11  "HMI force door close"
  B196:1/0  "Chute door is closed"
  B196:1/1  "control chute door"
  B196:1/13  "force box conveyor on"
  B196:3/0  "for hmi to continue production unlatched by hmi"
  HSC:0.0  "top"
  HSC:0.3/6  "Underflow interrupt"
  HSC:0.3/7  "Overflow interrupt"
  HSC:1.0  "bot"
  HSC:1.3/6  "Underflow interrupt"
  HSC:1.3/7  "Overflow interrupt"
  I7_TRAC  
  I:0.0/0  "Encoder Signal "A""
  I:0.0/1  "Encoder Signal "B""
  I:0.0/4  "Encoder Signal "A""
  I:0.0/5  "Encoder Signal "B""
  I:0.1/4  "not used"
  I:0.1/5  "not used"
  I:0.1/6  "not used"
  I:0.1/7  "not used"
  I:0.1/8  "not used"
  I:0.1/9  "not used"
  I:0.1/10  "not used"
  I:0.1/11  "not used"
  I:0.1/12  "not used"
  I:0.1/13  "not used"
  I:0.1/14  "not used"
  I:0.1/15  "not used"
  I:0.2  "not used"
  I:0.2/3  "Packaging Conveyor full"
  I:0.2/4  "Packaging Conveyor Box in Position"
  I:0.3  "not used"
  I:0.4  "Spare Analog Input 1"
  I:0.5  "Spare Analog Input 2"
  I:0.6  "Spare Analog Input 3"
  I:2.0/0  FRONT_ESTOP
  I:2.0/1  REAR_ESTOP
  I:2.0/8  FRONT_DOOR  "front door signal ce models only"
  I:2.0/9  REAR_DOOR  "rear door signal ce models only"
  I:2.0/11  "spare"
  L13:183  TKS_PER_SECOND
  L23:19  TOP_OPT_FAIL_CT
  L23:34  AIR_PRESSURE_FAULT
  L28:0  INS_1_TIME
  L29:0  INS_1_POS
  L30:0  INS_5_TIME
  L31:0  INS_5_POS
  L32:0  INS_6_TIME
  L33:0  INS_6_POS
  L192:1  BOT_LAST_TIME  "rtc bot belt previous movement event time"
  L192:2  BOT_CYCLE_TIME  "rtc bot belt time between events"
  L192:7  FROM_REAL  "distance from real part signal at optic location"
  L192:8  FROM_TRACKED  "distance from tracked part signal at optic location"
  L192:16  TOP_LAST_TIME  "rtc top belt previous movement event time"
  L192:17  TOP_CYCLE_TIME  "rtc top belt time between events"
  L199:5  ACQTM51
  L199:6  ACQTM52
  L199:7  ACQTM53
  L199:9  "ones"
  L199:10  "billions"
  L199:13  DUMP_LONG
  L199:15  ACQTM11
  L199:16  ACQTM12
  L199:17  ACQTM13
  L199:20  RESULTTM1
  L199:22  CLEARTIME5COUNT
  L199:23  CLEARTIME6COUNT
  L199:24  ACQTM61
  L199:25  ACQTM62
  L199:26  ACQTM63
  L199:27  TMSINCETRIG1
  L199:29  TMSINCETRIG5
  L199:30  TMSINCETRIG6
  L199:31  CLEARTIME1COUNT
  L199:32  RESULTTM5
  L199:33  RESULTTM6
  L199:34  MAXACQTM1
  L199:36  MAXACQTM6
  N7  
  N101:2  I3_TRIG_LOC
  N101:3  I4_TRIG_LOC
  O:0.0/1  "spare"
  O:0.0/11  "Spare"
  O:0.0/12  "not used"
  O:0.0/13  "not used"
  O:0.0/14  "not used"
  O:0.0/15  "not used"
  O:0.1  "not used"
  O:0.2  "not used"
  O:0.3  "not used"
  O:0.5  "spare analog output"
  O:3.0/0  "spare"
  O:3.0/2  "spare"
  O:3.0/3  "light curtain range selection /* needed? */"
  O:3.0/7  "door unlocks on CE models"
  O:3.0/8  "Light?"
  O:3.0/9  NUT_HOPPER  "Nut Hopper Enable"
  O:3.0/11  NUT_FEEDER_AIR  "Nut Feeder Bowl Air Enable"
  PFILE:6  "check for part jams"
  PFILE:10  "Bottom belt HSC"
  PFILE:12  "Top belt HSC"
  Q2:55  END_OF_MAIN
  Q5:94  END_OF_BELTS
  T20:0  "Trigger On Time"
  U:9  "slow data"
  U:24  "check skipped fail rate"
  U:28  "faults"
  U:29  "speed"
  U:30  "count"
  U:31  "rate calc"
  U:32  "boxer"
  U:33  "bulk pack"
  U:34  "customer boxing unit signals"
  U:35  "cleanup"

COMMENTS NOT ATTACHED TO A CURRENT RUNG
  R6:2: B41 is the top good 3 file
  R6:11/DN: B39 is the top good 2 file
  R6:10/DN: B37 is the top good 1 file
  R6:6/DN: B35 is the top NG file
  B100:1/15: what is this code for?
  R6:0: B36 is the bottom GOOD file
  R6:4: B34 is the bottom NG file
  R6:6: B35 is the top NG file
  R6:10: B37 is the top good 1 file

REVISION NOTES
  13: updated count reset
  14: added io moduals
  15: multiple steps toward new hmi integration
  21: test
  27: fix error if bulk pack and no boxing fallout were on

DATA TABLE (non-zero values as saved)
DATA B3
% B3:0 % 0X88A2 0X0141 0X4041 0XA101 0XC8BF 0X15D0 0X0430 0X0461 0X4FC0 0X2338
% B3:10 % 0X21E8 0X40C6 0X4000 0X1B32 0X0001 0X2000 0X0000 0X0000 0X0000 0X0000
% B3:20 % 0X0100 0X0000 0X0000 0X0000 0X0000 0X0000 0X0000 0X0000 0X0000 0X0000
% B3:50 % 0X0001 0X0000 0X0000 0X0000 0X0000 0X0000 0X0000 0X0000 0X0000 0X0000
DATA T4
% .PRE .ACC %
% T4:0 % 0 1
% T4:1 % 150 0
% T4:2 % 400 0
% T4:3 % 300 227
% T4:4 % 1000 0
% T4:5 % 5 5
% T4:6 % 10 10
% T4:7 % 150 0
% T4:8 % 20 11
% T4:9 % 50 9
% T4:10 % 200 200
% T4:11 % 400 0
% T4:12 % 80 81
% T4:13 % 250 0
% T4:14 % 666 0
% T4:15 % 1000 1004
% T4:16 % 400 0
% T4:17 % 100 52
% T4:18 % 5 0
% T4:19 % 300 0
% T4:20 % 200 0
% T4:21 % 200 0
% T4:22 % 200 0
% T4:23 % 250 0
% T4:24 % 666 0
% T4:25 % 666 0
% T4:26 % 666 0
% T4:27 % 250 0
% T4:28 % 250 0
% T4:29 % 5000 0
% T4:30 % 333 0
% T4:31 % 500 43
% T4:32 % 300 231
% T4:33 % 222 15
% T4:34 % 1111 0
% T4:35 % 23 0
% T4:36 % 5000 0
% T4:37 % 500 0
DATA C5
% .PRE .ACC %
% C5:0 % 32766 0
DATA R6
% .LEN .POS %
% R6:0 % 1250 0
% R6:1 % 16 0
% R6:2 % 1050 0
% R6:3 % 1050 0
% R6:4 % 1250 0
% R6:5 % 1250 0
% R6:6 % 1713 0
% R6:7 % 16 0
% R6:8 % 1024 0
% R6:9 % 3 0
% R6:10 % 1713 0
% R6:11 % 1050 0
% R6:12 % 10 0
% R6:13 % 10 0
% R6:14 % 10 0
% R6:15 % 10 0
% R6:16 % 1713 0
% R6:17 % 1713 0
% R6:18 % 1050 0
% R6:19 % 10 0
DATA N7
% N7:0 % 10 3 871 130 3 0 0 0 500 43
% N7:10 % 1000 43 0 8 22 22 1000 2000 50 1050
% N7:20 % 0 1329 16 2000 0 48 0 0 0 250
% N7:30 % 666 55 150 0 47 641 40 43 0 43
% N7:40 % 18 38 1 37 141 1211 682 1211 18 15
% N7:50 % 14 16 15 16 17 650 0 0 73 3
% N7:60 % 1713 1713 1050 3 73 160 4999 5 400 400
% N7:70 % 100 200 300 400 90 190 290 390 3 2
% N7:80 % 100 150 1268 1276 1271 1280 6 16 0 0
% N7:90 % 2011 4 4 12 1 6 16 4 250 12
% N7:100 % 1003 90 110 100 175 25 0 0 0 0
% N7:190 % -128 27477 27605 32767 0 0 0 0 0 0
DATA F8
% F8:0 % 6
DATA L13
% L13:0 % 148344 959262 0 125133 1463898
% L13:5 % 1 2704 333840227 611253 125133
% L13:10 % 125901 -1 0 15 90
% L13:15 % 577129669 -2147483648 2147483647 2147483647 82058
% L13:20 % 1118885267 -45793823 1200 0 100
% L13:25 % 150768 156084 137550 0 243269039
% L13:30 % 333859845 150822 1020000 243289470 700
% L13:35 % 0 126074 2724 942002793 942002824
% L13:40 % 0 1000000000 1000000 243289442 243299947
% L13:45 % 146615044 30 0 28 1117346621
% L13:50 % 333829768 333840273 243249531 0 0
% L13:55 % 203982 333837406 2082 82393203 358
% L13:60 % 132085 2319140 0 600 -1
% L13:65 % 100 -100 732972238 941960134 2
% L13:70 % 1117347141 160 8 0 1117346621
% L13:75 % 11 30 100 243292469 -1
% L13:80 % 557730 74 -74 40 208239
% L13:85 % 274296 5 0 0 333829800
% L13:90 % 203983 3 752580 5 243299972
% L13:95 % 679743587 176 0 146615070 6143
% L13:100 % 3400 524295 2100 1312119 176
% L13:105 % 6143 568360 1117346494 32 1117346488
% L13:110 % 6 180 0 -53301564 -53301568
% L13:115 % -53301561 7 4 -53301565 150726
% L13:120 % 32 46 54 0 85
% L13:125 % 0 1117347141 683000 3276501 274297
% L13:130 % 0 11 104 0 306
% L13:135 % 0 34 274296 1016 0
% L13:140 % 4 -4 36 0 0
% L13:145 % 333840366 5 333837499 5 8
% L13:150 % 1605500 67108884 46 -46 1
% L13:155 % 10 -10 0 32 5637628
% L13:160 % 7 25 26 132548 285213229
% L13:165 % -53301172 -63096029 -53301172 -63096029 1055291
% L13:170 % 143889 3306 2408314 800 400
% L13:175 % -1610612220 262148 537395242 536872983 268437542
% L13:180 % 732972238 0 0 1000000 0
% L13:185 % 0 0 942010207 0 50073
% L13:190 % 5000000 67108896 0 134217728 65536
% L13:195 % 2165248 138543120 10 -2147352060 1207976008
% L13:200 % 100671752 4481 536871424 805324800 168855553
% L13:205 % 0 2097152 524288 3030025 2008408
% L13:210 % -2111790848 4210696 4194320 65536 1048608
% L13:215 % 136314880 262145 35655680 1589280 0
% L13:220 % 16 0 4096 50332160 71303296
% L13:225 % 1073741824 1049600 1107296257 8192 -2113929216
% L13:230 % 33560576 256 1141374976 1024 -2147483584
% L13:235 % 0 270532608 8 262144 2
% L13:240 % 0 0 262144 65536 128
% L13:245 % 0 2097156 1024 268996608 -2071985920
% L13:250 % 16777216 2097152 262160 0 0
DATA L19
% L19:0 % 243271160 243271503 243272028 243272399 243280944
% L19:5 % 243281980 243282378 243282630 243285495 243285927
% L19:10 % 243288491 243290281 243290511 243295030 243298338
% L19:15 % 243269039 243270292 16777216 256 262144
% L19:20 % 4 0 0 0 0
% L19:25 % 0 1376256 4096 8 33652736
% L19:30 % 131072 524288 -2147483648 0 -2147483648
% L19:35 % 0 0 84 0 32768
% L19:40 % 0 4096 1073741824 0 0
% L19:45 % 256 0 0 16 5250
DATA L20
% L20:0 % 243287105 243287538 243290101 243291887 243292119
% L20:5 % 243296641 243299947 243180806 243181340 243181898
% L20:10 % 243183490 243184399 243184585 243184766 243185502
% L20:15 % 243186043 243186399 243187659 243188560 243188751
% L20:20 % 243189296 243190405 243191682 243195548 243195907
% L20:25 % 243196823 243198246 243198438 243200983 243201520
% L20:30 % 243202086 243202450 243203910 243207179 243207543
% L20:35 % 243207720 243212305 243213929 243215049 243215962
% L20:40 % 243217946 243219538 243220431 243221538 243221914
% L20:45 % 243222980 243226036 243226230 243227697 243228206
% L20:50 % 243228929 243229652 243230735 243230913 243232364
% L20:55 % 243232905 243233658 243234154 243238167 243238357
% L20:60 % 243239638 243239812 243241452 243242171 243242543
% L20:65 % 243242911 243243089 243244366 243244920 243245445
% L20:70 % 243245631 243245821 243247086 243247814 243249112
% L20:75 % 243253684 243254391 243254598 243257164 243259098
% L20:80 % 243259272 243260177 243261168 243261731 243262735
% L20:85 % 243263317 243263582 243263768 243264033 243268356
% L20:90 % 243270646 243271903 243272771 243273114 243273634
% L20:95 % 243274011 243282554 243283592 243283988 243284240
% L20:100 % 33554432 37224448 1073751040 536870914 0
% L20:105 % 0 1 1057 0 0
% L20:110 % 33554432 1024 0 0 0
% L20:115 % 0 0 134219777 112 1073741824
% L20:120 % 16777216 2097152 32896 1073752096 134479876
% L20:125 % 16512 32768 68157444 84934656 0
% L20:130 % 1073741824 12582912 67112960 536873088 67109120
% L20:135 % 772 67109008 4096 67108864 8408096
% L20:140 % 67108864 536891393 268435456 4194592 1048832
% L20:145 % 8390672 33024 2129920 33557056 268435456
% L20:150 % 268435456 262656 16777216 0 10
% L20:155 % 32768 1 0 1048960 0
% L20:160 % 134217728 0 0 134217728 16777472
% L20:165 % 524352 0 1 0 131072
% L20:170 % 536870912 2195457 0 262144 0
% L20:175 % 65536 0 268435456 16384 1048576
% L20:180 % 0 16 0 0 1073743872
% L20:185 % 4456448 0 67108880 75497472 16384
% L20:190 % 512 -2013265920 131106 -2147463168 -2112880640
% L20:195 % 4098 84017472 2101780 8 272761088
% L20:200 % 514 67109376 67141632 0 2048
% L20:205 % 536870912 67108864 32768 0 2
% L20:210 % 8650752 0 16 8388608 0
% L20:215 % -2147482624 134217728 8 16384 0
% L20:220 % 67108866 1074268160 0 32 -2139095040
% L20:225 % 16777216 256 67108864 4194320 2048
% L20:230 % 272630016 0 1073774592 -2147483644 4
% L20:235 % 3146304 8262 65600 16777344 262144
% L20:240 % 1024 134217728 68 4160 1073750528
% L20:245 % 1073741824 268500992 0 285212676 824184832
% L20:250 % 4096 262400 134219776 8192 4096
% L20:255 % 1073774592
DATA L21
% L21:0 % -53304278 -53304173 -53303553 -53303121 -53303065
% L21:5 % -53301971 -53301172 -53329993 -53329864 -53329729
% L21:10 % -53329344 -53329124 -53329079 -53329035 -53328857
% L21:15 % -53328726 -53328640 -53328335 -53328117 -53328071
% L21:20 % -53327939 -53327671 -53327362 -53326428 -53326341
% L21:25 % -53326120 -53325776 -53325730 -53325115 -53324985
% L21:30 % -53324848 -53324760 -53324407 -53323616 -53323528
% L21:35 % -53323485 -53322376 -53321983 -53321712 -53321491
% L21:40 % -53321011 -53320626 -53320410 -53320142 -53320051
% L21:45 % -53319793 -53319054 -53319007 -53318652 -53318529
% L21:50 % -53318354 -53318179 -53317917 -53317874 -53317523
% L21:55 % -53317392 -53317210 -53317090 -53316119 -53316073
% L21:60 % -53315763 -53315721 -53315324 -53315150 -53315060
% L21:65 % -53314971 -53314928 -53314619 -53314485 -53314358
% L21:70 % -53314313 -53314267 -53313961 -53313785 -53313471
% L21:75 % -53312365 -53312194 -53312144 -53311523 -53311055
% L21:80 % -53311013 -53310794 -53310554 -53310418 -53310175
% L21:85 % -53310034 -53309970 -53309925 -53309861 -53308815
% L21:90 % -53308261 -53307957 -53307747 -53307664 -53307538
% L21:95 % -53307447 -53305379 -53305128 -53305032 -53304971
% L21:100 % 32 83886080 1094746112 20480 -2143289344
% L21:105 % 1073741856 65536 0 4174 543162960
% L21:110 % 263274 4224 67108872 134479872 -2147479472
% L21:115 % 536870912 39168 364544 149512 18564
% L21:120 % 1127432 537395200 268352 67109384 1024
% L21:125 % 4096 -2147483648 1 131072 1
% L21:130 % 8 1048576 0 -2139094080 18875272
% L21:135 % 416 7425 603981440 67110528 138016
% L21:140 % 33556096 1073749014 5776064 50355200 39488
% L21:145 % 8814849 8478720 -2147106560 -2012807168 3671296
% L21:150 % 5390464 2752512 20971553 532480 1078722560
% L21:155 % 128 33554433 1024 4196360 1344012289
% L21:160 % 1207959872 8429584 33554435 1080033282 656128
% L21:165 % 268435456 524352 -2139094008 704692248 134218020
% L21:170 % 134225924 0 704512 -2147445760 43008
% L21:175 % 134294528 32 1073741832 2097286 1049088
% L21:180 % 16908968 101711874 131072 10756096 1073774740
% L21:185 % 33554688 786560 0 135204 50364416
% L21:190 % 33554496 -1609562624 268456960 262144 8192
% L21:195 % 1073741824 268435456 131072 0 524808
% L21:200 % 2097152 2097152 2432 0 1048576
% L21:205 % 16777728 526688 67108880 5378080 8704
% L21:210 % 33554432 2097153 4366336 704718849 36131460
% L21:215 % 1572864 1266698272 12583040 -1555038208 18690
% L21:220 % 512 134217876 1073872896 5120 1073741824
% L21:225 % 0 335609920 16 -2147483646 524288
% L21:230 % 68157472 80 4194304 134221824 67109248
% L21:235 % 134217728 134217728 537952256 603979776 16387
% L21:240 % 2949269 688128 1494239520 4194304 38535172
% L21:245 % 1073742226 33587348 67125289 2048 536870912
% L21:250 % -2147466238 65536 1879261186 67108931 5507744
% L21:255 % 1
DATA L22
% L22:0 % 75768173 75768404 142529185 143026808 143427984
% L22:5 % 143428215 143428445 143428675 143428903 143429134
% L22:10 % 143429361 143429592 143429821 143430050 144170464
% L22:15 % 144206730 146615044 74246159 74246583 74248049
% L22:20 % 74248302 74248688 74250474 74251356 74251587
% L22:25 % 74252336 74256349 74256801 74260152 74260543
% L22:30 % 74261319 74262103 74262384 74265850 74270960
% L22:35 % 74274708 74275809 74285933 74288281 74288854
% L22:40 % 74311814 74312195 75766344 75766572 75766801
% L22:45 % 75767030 75767260 75767487 75767717 75767945
DATA L23
% L23:0 % -65222797 -65222755 -64084516 -63964129 -63867075
% L23:5 % -63867019 -63866963 -63866907 -63866852 -63866796
% L23:10 % -63866741 -63866686 -63866630 -63866575 -63687448
% L23:15 % -63678674 -63096029 -65498962 -65498885 -65498619
% L23:20 % -65498573 -65498503 -65498179 -65498019 -65497977
% L23:25 % -65497841 -65497113 -65497031 -65496423 -65496352
% L23:30 % -65496211 -65496069 -65496018 -65495389 -65494462
% L23:35 % -65493782 -65493582 -65491745 -65491319 -65491215
% L23:40 % -65487049 -65486980 -65223129 -65223088 -65223046
% L23:45 % -65223004 -65222963 -65222922 -65222880 -65222838
DATA L30
% L30:0 % 243260524 243260713 243260950 243261407 243261650
% L30:5 % 243261866 243262102 243262266 243262436 243262606
% L30:10 % 243262784 243262961 243263131 243263308 243263507
% L30:15 % 243263699 243264384 243265185 243265460 243265838
% L30:20 % 243266031 243266985 243272050 243272237 243272462
% L30:25 % 243272662 243272888 243273086 243273273 243273492
% L30:30 % 243273734 243276427 243276609 243276851 243277044
% L30:35 % 243278752 243279387 243279602 243281389 243281616
% L30:40 % 243285698 243286139 243289266 243289442 243258469
% L30:45 % 243258710 243258892 243259637 243260145 243260325
DATA L31
% L31:0 % 1117341374 1117341408 1117341451 1117341534 1117341578
% L31:5 % 1117341617 1117341660 1117341690 1117341721 1117341752
% L31:10 % 1117341784 1117341816 1117341847 1117341879 1117341915
% L31:15 % 1117341950 1117342074 1117342219 1117342269 1117342338
% L31:20 % 1117342373 1117342546 1117343465 1117343499 1117343540
% L31:25 % 1117343576 1117343617 1117343653 1117343687 1117343727
% L31:30 % 1117343771 1117344259 1117344292 1117344336 1117344371
% L31:35 % 1117344681 1117344796 1117344835 1117345160 1117345201
% L31:40 % 1117345942 1117346022 1117346589 1117346621 1117341001
% L31:45 % 1117341045 1117341078 1117341213 1117341305 1117341338
DATA L32
% L32:0 % 243266372 243268048 243268325 243268705 243268898
% L32:5 % 243274916 243275953 243276361 243276604 243279475
% L32:10 % 243279717 243279910 243282463 243284257 243284482
% L32:15 % 243289006 243292133 243292309 243249531 243249878
% L32:20 % 243250603 243251127 243251458 243251634 243251811
% L32:25 % 243252264 243252539 243253357 243253533 243254095
% L32:30 % 243255095 243255685 243255943 243256125 243256396
% L32:35 % 243257935 243258599 243258864 243260012 243260518
% L32:40 % 243260718 243261336 243263010 243263816 243264274
% L32:45 % 243264731 243265136 243265476 243265828 243265999
DATA L33
% L33:0 % 1117342435 1117342739 1117342789 1117342858 1117342893
% L33:5 % 1117343985 1117344173 1117344247 1117344291 1117344812
% L33:10 % 1117344856 1117344891 1117345355 1117345680 1117345721
% L33:15 % 1117346542 1117347109 1117347141 1117339379 1117339442
% L33:20 % 1117339574 1117339669 1117339729 1117339761 1117339793
% L33:25 % 1117339875 1117339925 1117340073 1117340105 1117340207
% L33:30 % 1117340389 1117340496 1117340543 1117340576 1117340625
% L33:35 % 1117340904 1117341025 1117341073 1117341281 1117341373
% L33:40 % 1117341409 1117341521 1117341825 1117341971 1117342054
% L33:45 % 1117342137 1117342210 1117342272 1117342336 1117342367
DATA B34
% B34:80 % 0X0200 0X0800 0X0000 0X4000 0X0040 0X5000 0X0000 0X0000 0X0100 0X8000
% B34:90 % 0X0080 0X0000 0X8400 0X0000 0X0000 0X8000 0X0000 0X0000 0X4000 0X0000
% B34:100 % 0X0000 0X0000 0X8000 0X0000 0X0000 0X0002 0X0000 0X0000 0X0000 0X0200
% B34:110 % 0X0000 0X0400 0X0000 0X0000 0X0000 0X0000 0X0220 0X0000 0X0100 0X0000
% B34:120 % 0X0000 0X0000 0X0000 0X1000 0X0000 0X0000 0X0000 0X8020
DATA B35
% B35:110 % 0X0000 0X0000 0X0200 0X0000 0X0000 0X0000 0X0000 0X0000 0X0000 0X0000
DATA B37
% B37:0 % 0X0000 0X0000 0X2000 0X0000 0X0000 0X0000 0X0000 0X0000 0X0000 0X0000
DATA B40
% B40:0 % 0XAAAA
DATA B41
% B41:50 % 0X0000 0X0000 0X0000 0X0000 0X1FC0 0X0000 0X0000 0X0000 0X0000 0X0000
DATA B100
% B100:0 % 0X8700 0X88A0 0X0004 0X0000 0X0000 0X0000 0X0000 0X0000 0X0000 0X0000
DATA N101
% N101:0 % 130 650 0 0 1166 100 867 1200 1200 1260
% N101:10 % 1269 1627 10 16055 655 20314 3110 300 333 500
% N101:20 % 1000 500 400 0 0 0 222 300 0 0
DATA L102
% L102:0 % 80 10 1 102 0
% L102:5 % 100 0 3 0 0
% L102:10 % -1 1194 0 0 752580
% L102:15 % 0 30 18 30 19
% L102:20 % 26 8 0 0 25
% L102:25 % 28 3407 34 525 19
% L102:30 % 160 2196 21 0 12
% L102:35 % 51 6000 0 999999 26
% L102:40 % 0 4 0 0 3
